{attribute 'linkalways'} 
{attribute 'no_explicit_call' := 'This FB is a CLASS and must be accessed using methods or properties'}
{attribute 'enable_dynamic_creation'}
FUNCTION_BLOCK FINAL FRAC_LREAL EXTENDS Node
VAR
	in : _LREAL(0.0);
	out : _LREAL(0.0);
END_VAR

METHOD PUBLIC Clone : I_Node
VAR
	pNode : POINTER TO FRAC_LREAL;
END_VAR
pNode := __NEW(FRAC_LREAL);
Clone := pNode^;
END_METHOD

METHOD FB_init : BOOL
VAR_INPUT
	bInitRetains : BOOL; // if TRUE, the retain variables are initialized (warm start / cold start)
	bInCopyCode : BOOL;  // if TRUE, the instance afterwards gets moved into the copy code (online change)
END_VAR
AddInput('in',THIS^.in);
AddOutput('out', THIS^.out);
END_METHOD

METHOD PROTECTED OnExecute
VAR
END_VAR
out.Value := FRAC(in.Value);
END_METHOD

END_FUNCTION_BLOCK

(* stored: Version 1.1.0.1, ProductVersion 3.1.4024.15
   POU FRAC_LREAL: Id {c3be8d02-3bea-44a4-b5cf-aa1e5513a012}, SpecialFunc None
   Folder Constructor: Id {bb9edb0c-81e9-421f-ad58-ff8d77b5588a}
   Method Clone: Id {28befac4-deb8-4c3f-8ba3-be28cf72927c}
   Method FB_init: Id {b2c91e03-b106-4e07-ab76-20d8eff2488e}
   Method OnExecute: Id {cd292fbb-bd3e-4ad3-8a88-49c62370d857} *)
